// TIA Portal project "Project1" (V17)

(* hardware
DEVICE "S7-1200 station_1"  S7-1200 Station
   slot 0: "Rack_0"  S7-1200 Rack  Rack  V1.0
   slot 1: "PLC_1"  CPU 1212C DC/DC/DC  6ES7 212-1AE40-0XB0  V4.5
*)

// ===== PLC "PLC_1"  CPU 1212C DC/DC/DC =====

VAR_GLOBAL   // PLC tag table "Default tag table"
   "System_Byte" AT %MB1 : Byte;
   "FirstScan" AT %M1.0 : Bool;
   "DiagStatusUpdate" AT %M1.1 : Bool;
   "AlwaysTRUE" AT %M1.2 : Bool;
   "AlwaysFALSE" AT %M1.3 : Bool;
   "Clock_Byte" AT %MB0 : Byte;
   "Clock_10Hz" AT %M0.0 : Bool;
   "Clock_5Hz" AT %M0.1 : Bool;
   "Clock_2.5Hz" AT %M0.2 : Bool;
   "Clock_2Hz" AT %M0.3 : Bool;
   "Clock_1.25Hz" AT %M0.4 : Bool;
   "Clock_1Hz" AT %M0.5 : Bool;
   "Clock_0.625Hz" AT %M0.6 : Bool;
   "Clock_0.5Hz" AT %M0.7 : Bool;
   "Pallet at entry" AT %I62.0 : Bool;
   "Pallet at exit" AT %I62.1 : Bool;
   "Pallet loaded" AT %I62.2 : Bool;
   "Box at entry" AT %I62.3 : Bool;
   "Pusher limit" AT %I62.4 : Bool;
   "Plate limit" AT %I62.5 : Bool;
   "Clamped" AT %I62.6 : Bool;
   "Pallet feeder" AT %Q62.7 : Bool;
   "Load pallet" AT %Q62.6 : Bool;
   "Exit conveyor" AT %Q62.5 : Bool;
   "Move to limit" AT %Q62.4 : Bool;
   "Elevator up" AT %Q62.3 : Bool;
   "Box feeder" AT %Q62.2 : Bool;
   "Turn" AT %Q62.0 : Bool;
   "Push" AT %Q61.7 : Bool;
   "Load belt" AT %Q61.6 : Bool;
   "Clamp" AT %Q61.5 : Bool;
   "Open plate" AT %Q61.4 : Bool;
   "Warning light" AT %Q61.3 : Bool;
   "Start light" AT %Q61.2 : Bool;
   "Reset light" AT %Q61.1 : Bool;
   "Stop light" AT %Q61.0 : Bool;
   "Elevator moving" AT %I62.7 : Bool;
   "Start" AT %I63.0 : Bool;
   "Stop" AT %I63.1 : Bool;
   "Reset" AT %I63.2 : Bool;
   "Sitema ligado" AT %M10.0 : Bool;
   "Elevator down" AT %Q62.1 : Bool;
   "Parts emitter" AT %Q60.0 : Bool;
   "Sitema em espera" AT %M10.1 : Bool;
   "Reset CTU" AT %M10.2 : Bool;
   "Push n" AT %M100.0 : Bool;
   "push reset" AT %M10.3 : Bool;
   "push limiter p" AT %M100.1 : Bool;
   "Pallet feito" AT %M10.4 : Bool;
   "clamped merory N" AT %M100.2 : Bool;
   "Clamped reset" AT %M10.5 : Bool;
   "Pallet feito reset" AT %M10.6 : Bool;
   "limit plate memory P" AT %M100.3 : Bool;
   "Plate limit reset" AT %M10.7 : Bool;
   "Pallet emitter" AT %Q60.1 : Bool;
END_VAR

// folder: System blocks/Program resources

DATA_BLOCK "IEC_Counter_0_DB"   // DB1
{ S7_Optimized_Access := 'TRUE' }
AUTHOR : Simatic
FAMILY : IEC
NAME : CNTR
VERSION : 1.0
// stored: InstanceOfName IEC_COUNTER
"IEC_COUNTER"
BEGIN
END_DATA_BLOCK

DATA_BLOCK "IEC_Timer_0_DB"   // DB2
{ S7_Optimized_Access := 'TRUE' }
AUTHOR : Simatic
FAMILY : IEC
NAME : IEC_TMR
VERSION : 1.0
// stored: InstanceOfName IEC_TIMER
"IEC_TIMER"
BEGIN
END_DATA_BLOCK

DATA_BLOCK "IEC_Counter_0_DB_1"   // DB3
{ S7_Optimized_Access := 'TRUE' }
AUTHOR : Simatic
FAMILY : IEC
NAME : CNTR
VERSION : 1.0
// stored: InstanceOfName IEC_COUNTER
"IEC_COUNTER"
BEGIN
END_DATA_BLOCK

DATA_BLOCK "IEC_Timer_0_DB_1"   // DB4
{ S7_Optimized_Access := 'TRUE' }
AUTHOR : Simatic
FAMILY : IEC
NAME : IEC_TMR
VERSION : 1.0
// stored: InstanceOfName IEC_TIMER
"IEC_TIMER"
BEGIN
END_DATA_BLOCK

DATA_BLOCK "IEC_Timer_0_DB_2"   // DB5
{ S7_Optimized_Access := 'TRUE' }
AUTHOR : Simatic
FAMILY : IEC
NAME : IEC_TMR
VERSION : 1.0
// stored: InstanceOfName IEC_TIMER
"IEC_TIMER"
BEGIN
END_DATA_BLOCK

DATA_BLOCK "IEC_Timer_0_DB_3"   // DB6
{ S7_Optimized_Access := 'TRUE' }
AUTHOR : Simatic
FAMILY : IEC
NAME : IEC_TMR
VERSION : 1.0
// stored: InstanceOfName IEC_TIMER
"IEC_TIMER"
BEGIN
END_DATA_BLOCK

// folder: (top level)

FUNCTION "MHJ-PLC-Lab-Function-S71200" : Void   // FC9000, SCL
{ S7_Optimized_Access := 'TRUE' }
VERSION : 0.1
   VAR_TEMP
      rdTimeReturn : Int;
      outputTime : DTL;
      SyncVal : Byte;
      forVal : Int;
      forVal_2 : Int;
      Value : Byte;
   END_VAR
   VAR CONSTANT
      CompVal : Byte := 16#34;
      Value_01 : Byte := 16#11;
      Value_01_DW : DWord := 16#A165_D992;
      Value_02_DW : DWord := 16#58BE_4401;
   END_VAR
BEGIN

   #Value:=PEEK(area := 16#82,
        dbNumber := 0,
        byteOffset := 511);
   #Value := #Value + 1;

   POKE(area := 16#82,
        dbNumber := 0,
        byteOffset := 511,
        value := #Value);

   POKE(area:=16#81,
        dbNumber:=0,
        byteOffset:=1016,
        value:=#Value_01_DW);
   POKE(area := 16#81,
        dbNumber := 0,
        byteOffset := 1020,
        value := #Value_02_DW);

   POKE(area := 16#81,
        dbNumber := 0,
        byteOffset := 511,
        value := B#16#00);

   FOR #forVal := 0 TO 120 DO
       FOR #forVal_2:=0 TO 10 DO
           #rdTimeReturn:=RD_SYS_T(#outputTime);
           #rdTimeReturn := WR_SYS_T(#outputTime);
           #rdTimeReturn := RD_SYS_T(#outputTime);
           #rdTimeReturn := WR_SYS_T(#outputTime);
       END_FOR;
       #SyncVal:= PEEK(area := 16#81,
                      dbNumber := 0,
                      byteOffset := 511);
       IF #SyncVal = #CompVal THEN
          GOTO M_1;
       END_IF;
   END_FOR;
   RETURN;

   M_1:
   POKE(area := 16#81,
        dbNumber := 0,
        byteOffset := 511,
        value := B#16#0);
END_FUNCTION

ORGANIZATION_BLOCK "Main"   // OB1, LAD, ProgramCycle
TITLE = "Main Program Sweep (Cycle)"
{ S7_Optimized_Access := 'TRUE' }
VERSION : 0.1
   VAR_INPUT
      Initial_Call : Bool;   // Initial call of this OB
      Remanence : Bool;   // =True, if remanent data are available
   END_VAR
   VAR_TEMP   // added for the SCL form of the ladder/FBD networks
      _w1 : Bool;
      _w2 : Bool;
   END_VAR
BEGIN

REGION Network 1
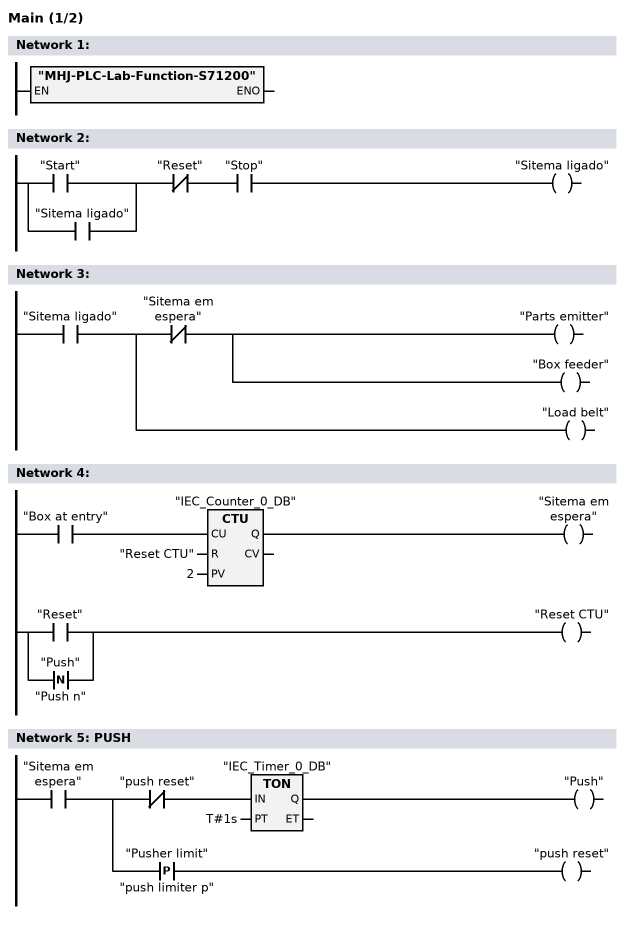
   RUNG wire#powerrail
      "MHJ-PLC-Lab-Function-S71200"()
   END_RUNG
   // the same network as SCL:
   "MHJ-PLC-Lab-Function-S71200"();
END_REGION

REGION Network 2
   RUNG wire#powerrail
      Contact( "Start" )
      wire#w1
      I_Contact( "Reset" )
      Contact( "Stop" )
      Coil( "Sitema ligado" )
   END_RUNG
   RUNG wire#powerrail
      Contact( "Sitema ligado" )
   END_RUNG wire#w1
   // the same network as SCL:
   "Sitema ligado" := ("Start" OR "Sitema ligado") AND NOT "Reset" AND "Stop";
END_REGION

REGION Network 3
   RUNG wire#powerrail
      Contact( "Sitema ligado" )
      wire#w1
      I_Contact( "Sitema em espera" )
      wire#w2
      Coil( "Parts emitter" )
   END_RUNG
   RUNG wire#w2
      Coil( "Box feeder" )
   END_RUNG
   RUNG wire#w1
      Coil( "Load belt" )
   END_RUNG
   // the same network as SCL:
   "Parts emitter" := "Sitema ligado" AND NOT "Sitema em espera";
   "Box feeder" := "Parts emitter";
   "Load belt" := "Sitema ligado";
END_REGION

REGION Network 4
   "IEC_Counter_0_DB".CTU(CU := "Box at entry", R := "Reset CTU", PV := 2);
   "Sitema em espera" := "IEC_Counter_0_DB".Q;
   #_w1 := NOT "Push" AND "Push n";   // falling edge of "Push"
   "Push n" := "Push";
   "Reset CTU" := "Reset" OR #_w1;
END_REGION

REGION Network 5: PUSH
   "IEC_Timer_0_DB".TON(IN := "Sitema em espera" AND NOT "push reset", PT := T#1s);
   "Push" := "IEC_Timer_0_DB".Q;
   #_w1 := "Sitema em espera" AND "Pusher limit" AND NOT "push limiter p";   // rising edge of "Pusher limit"
   "push limiter p" := "Pusher limit";
   "push reset" := #_w1;
END_REGION

REGION Network 6: CLAMP
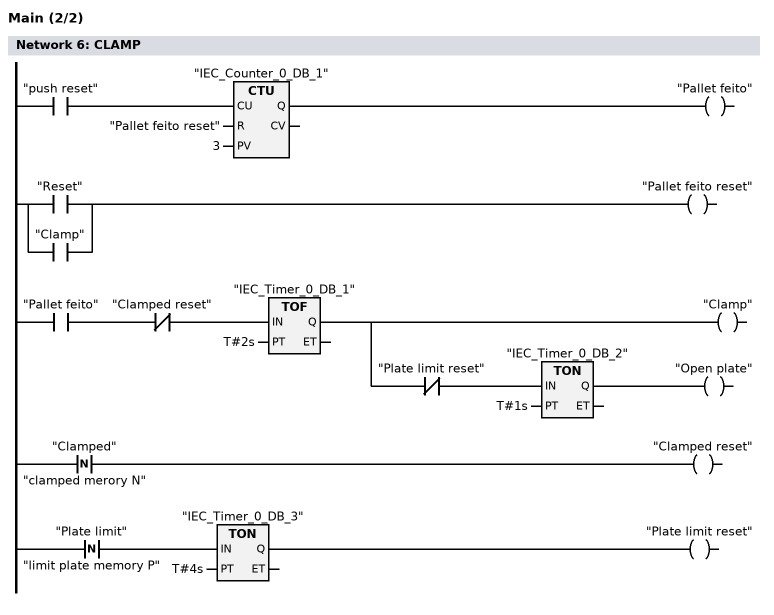
   "IEC_Counter_0_DB_1".CTU(CU := "push reset", R := "Pallet feito reset", PV := 3);
   "Pallet feito" := "IEC_Counter_0_DB_1".Q;
   "Pallet feito reset" := "Reset" OR "Clamp";
   "IEC_Timer_0_DB_1".TOF(IN := "Pallet feito" AND NOT "Clamped reset", PT := T#2s);
   "Clamp" := "IEC_Timer_0_DB_1".Q;
   "IEC_Timer_0_DB_2".TON(IN := "IEC_Timer_0_DB_1".Q AND NOT "Plate limit reset", PT := T#1s);
   "Open plate" := "IEC_Timer_0_DB_2".Q;
   #_w1 := NOT "Clamped" AND "clamped merory N";   // falling edge of "Clamped"
   "clamped merory N" := "Clamped";
   "Clamped reset" := #_w1;
   #_w2 := NOT "Plate limit" AND "limit plate memory P";   // falling edge of "Plate limit"
   "limit plate memory P" := "Plate limit";
   "IEC_Timer_0_DB_3".TON(IN := #_w2, PT := T#4s);
   "Plate limit reset" := "IEC_Timer_0_DB_3".Q;
END_REGION
END_ORGANIZATION_BLOCK